// TIA Portal project "Tangki" (V15.1)

(* hardware
DEVICE "S7-1200 station_1"  S7-1200 Station
   slot 0: "Rack_0"  S7-1200 Rack  Rack  V1.0
   slot 1: "PLC_1"  CPU 1214C AC/DC/Rly  6ES7 214-1BG40-0XB0  V4.2
   slot 3: "AQ 1x12BIT_1"  AQ1 signal board  6ES7 232-4HA30-0XB0  V1.0
DEVICE "HMI_1"  KTP700 Basic PN
   slot 0: "HMI_1"  KTP700 Basic PN  6AV2 123-2GB03-0AX0  15.1.0.0
   slot 1: "HMI_RT_1"  KTP700 Basic PN  6AV2 123-2GB03-0AX0  15.1.0.0
   slot 5: "HMI_1.IE_CP_1"  PROFINET Interface  15.0.1.0
      slot 1: "PROFINET Interface_1"  PROFINET Interface
         slot 1: "Port_1"  Port
DEVICE "PC station"  SIMATIC PC station
   slot 0: "PC station"  Rail  SIMATIC PC-Station  V1.0
      slot 125: "Stationmanager"  Station_Manager  V6.0.4
   slot 1: "IE general_1"  IE General  IE_CP  V8.2.0
   slot 2: "HMI_RT_2"  WinCC RT Advanced  6AV2 104-0xxxx-xxxx  15.1.0.0
      slot 33792: "Host interface"  Host interface
*)

// ===== PLC "PLC_1"  CPU 1214C AC/DC/Rly =====

VAR_GLOBAL   // PLC tag table "Default tag table"
   "Start" AT %I0.0 : Bool;
   "Stop" AT %I0.1 : Bool;
   "Analog" AT %IW64 : Int;
   "Auto" AT %I1.0 : Bool;
   "Motor_ON" AT %Q0.0 : Bool;
   "HMI_Start" AT %M0.0 : Bool;
   "HMI_Stop" AT %M0.1 : Bool;
   "ON" AT %M0.2 : Bool;
   "Motor_OFF" AT %M0.3 : Bool;
   "wkwkk" AT %M0.4 : Bool;
   "SCADA_START" AT %M0.5 : Bool;
   "SCADA_OFF" AT %M0.6 : Bool;
   "ibnu" AT %M0.7 : Bool;
   "off" AT %M1.0 : Bool;
   "Motor_nyala" AT %M1.1 : Bool;
END_VAR

DATA_BLOCK "Data_block_1"   // DB1
{ S7_Optimized_Access := 'TRUE' }
VERSION : 0.1
   VAR
      Scal1 : Real;
      ACT : Real;
   END_VAR
BEGIN
END_DATA_BLOCK

ORGANIZATION_BLOCK "Main"   // OB1, LAD, ProgramCycle
TITLE = "Main Program Sweep (Cycle)"
{ S7_Optimized_Access := 'TRUE' }
VERSION : 0.1
   VAR_INPUT
      Initial_Call : Bool;   // Initial call of this OB
      Remanence : Bool;   // =True, if remanent data are available
   END_VAR
BEGIN

REGION Network 1
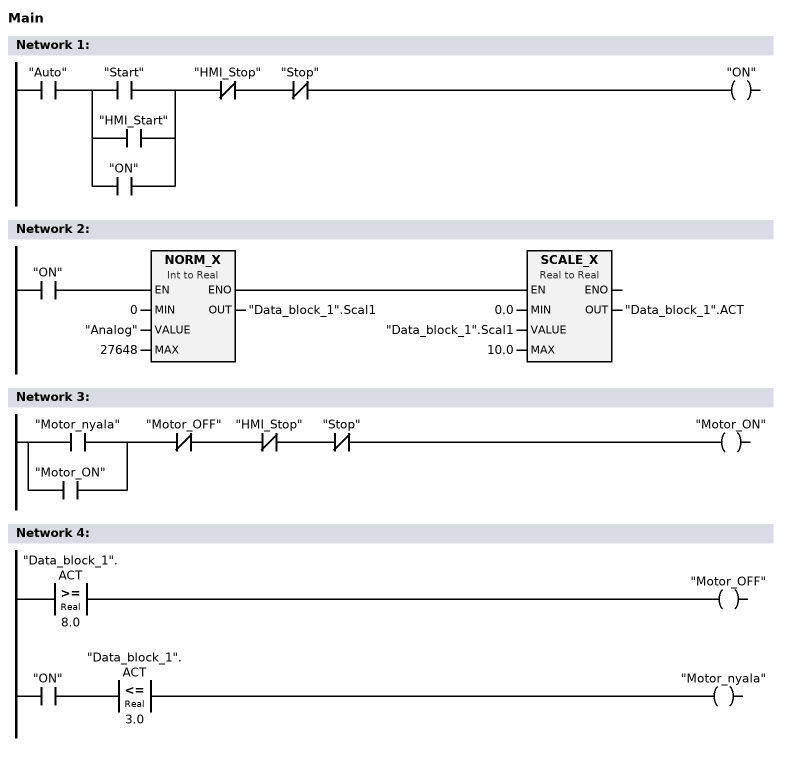
   RUNG wire#powerrail
      Contact( "Auto" )
      wire#w1
      Contact( "Start" )
      wire#w2
      I_Contact( "HMI_Stop" )
      I_Contact( "Stop" )
      Coil( "ON" )
   END_RUNG
   RUNG wire#w1
      Contact( "HMI_Start" )
   END_RUNG wire#w2
   RUNG wire#w1
      Contact( "ON" )
   END_RUNG wire#w2
   // the same network as SCL:
   "ON" := "Auto" AND ("Start" OR "HMI_Start" OR "ON") AND NOT "HMI_Stop" AND NOT "Stop";
END_REGION

REGION Network 2
   RUNG wire#powerrail
      Contact( "ON" )
      { S7_Templates := "[SrcType := Int, DestType := Real]" } Normalize(min := 0, value := "Analog", max := 27648, out => "Data_block_1".Scal1)
      { S7_Templates := "[SrcType := Real, DestType := Real]" } Scale(min := 0.0, value := "Data_block_1".Scal1, max := 10.0, out => "Data_block_1".ACT)
   END_RUNG
   // the same network as SCL:
   IF "ON" THEN
       "Data_block_1".Scal1 := NORM_X(MIN := 0, VALUE := "Analog", MAX := 27648);
       "Data_block_1".ACT := SCALE_X(MIN := 0.0, VALUE := "Data_block_1".Scal1, MAX := 10.0);
   END_IF;
END_REGION

REGION Network 3
   RUNG wire#powerrail
      Contact( "Motor_nyala" )
      wire#w1
      I_Contact( "Motor_OFF" )
      I_Contact( "HMI_Stop" )
      I_Contact( "Stop" )
      Coil( "Motor_ON" )
   END_RUNG
   RUNG wire#powerrail
      Contact( "Motor_ON" )
   END_RUNG wire#w1
   // the same network as SCL:
   "Motor_ON" := ("Motor_nyala" OR "Motor_ON") AND NOT "Motor_OFF" AND NOT "HMI_Stop" AND NOT "Stop";
END_REGION

REGION Network 4
   RUNG wire#powerrail
      { S7_Templates := "SrcType := Real" } GE_Contact(in1 := "Data_block_1".ACT, in2 := 8.0)
      Coil( "Motor_OFF" )
   END_RUNG
   RUNG wire#powerrail
      Contact( "ON" )
      { S7_Templates := "SrcType := Real" } LE_Contact(in1 := "Data_block_1".ACT, in2 := 3.0)
      Coil( "Motor_nyala" )
   END_RUNG
   // the same network as SCL:
   "Motor_OFF" := "Data_block_1".ACT >= 8.0;
   "Motor_nyala" := "ON" AND ("Data_block_1".ACT <= 3.0);
END_REGION
END_ORGANIZATION_BLOCK

(* ===== HMI "HMI_RT_1" =====
system functions are stored by id; their names below are inferred from use
connection "HMI_Connection_1": ETHERNET, SMART_S7_1200_OMS

HMI tags "Default tag table"
   "Motor_ON" : Bool = PLC Motor_ON AT %Q0.0, 1 s
   "HMI_Start" : Bool = PLC HMI_Start AT %M0.0, 1 s
   "HMI_Stop" : Bool = PLC HMI_Stop AT %M0.1, 1 s
   "Data_block_1_ACT" : Real = PLC Data_block_1.ACT, 1 s
   "Start" : Bool = PLC Start AT %I0.0, 1 s
   "Stop" : Bool = PLC Stop AT %I0.1, 1 s

screen "Screen_1" 800x480
   Button "Button_1" at 64,119 size 160x54; TextOff 'HMI START'
      on Press: SetBit("HMI_Start")
      on Release: ResetBit("HMI_Start")
      Appearance <- "HMI_Start"
   Circle "Circle_1" at 716,20 size 62x62
      Appearance <- "Motor_ON"
   Bar "Bar_1" at 566,80 size 115x260; MinimumValue 0; MaximumValue 10
      ProcessValue <- "Data_block_1_ACT"
   Button "Button_2" at 64,199 size 160x54; TextOff 'HMI STOP'
      on Release: ResetBit("HMI_Stop")
      on Press: SetBit("HMI_Stop")
      Appearance <- "HMI_Stop"
*)

(* ===== HMI "HMI_RT_2" =====
system functions are stored by id; their names below are inferred from use
connection "HMI_Connection_2": ETHERNET, S7_1200_OMS

HMI tags "Default tag table"
   "Motor_ON" : Bool = PLC Motor_ON AT %Q0.0, 1 s
   "HMI_Start" : Bool = PLC HMI_Start AT %M0.0, 1 s
   "HMI_Stop" : Bool = PLC HMI_Stop AT %M0.1, 1 s
   "Data_block_1_ACT" : Real = PLC Data_block_1.ACT, 1 s
   "SCADA_START" : Bool = PLC SCADA_START AT %M0.5, 1 s
   "SCADA_OFF" : Bool = PLC SCADA_OFF AT %M0.6, 1 s

screen "Screen_1" 1024x768
   Button "Button_1" at 182,144 size 123x51; TextOff 'SCADA ON'
      on Press: SetBit("HMI_Start")
      on Release: ResetBit("HMI_Start")
      Appearance <- "HMI_Start"
   Circle "Circle_1" at 681,60 size 91x91
      Appearance <- "Motor_ON"
   Bar "Bar_1" at 581,127 size 80x230; MinimumValue 0; MaximumValue 10
      ProcessValue <- "Data_block_1_ACT"
   Button "Button_2" at 182,210 size 123x51; TextOff 'SCADA OFF'
      on Release: ResetBit("HMI_Stop")
      on Press: SetBit("HMI_Stop")
      Appearance <- "HMI_Stop"
*)